FUNCTION INITIALIZE : BOOL
VAR_INPUT
END_VAR
VAR
	i : INT;
	GVL_IO: INT;
	SECTION2_DIG_INPUTS: INT;
	SECTION1_DIG_INPUTS: INT;
	JBOX_JBOX_GVL_LOGS: INT;
	NUM_TESTS_LOGGED: INT;
END_VAR


JBOX_GVL_LOGS.NUM_TESTS_LOGGED := 0;


JBOX_GVL_IO.SECTION1_DIG_INPUTS[0] := ADR(JBOX_GVL_IO.J7_24V_Up);
JBOX_GVL_IO.SECTION1_DIG_INPUTS[1] := ADR(JBOX_GVL_IO.J7_24V_Us);
JBOX_GVL_IO.SECTION1_DIG_INPUTS[2] := ADR(JBOX_GVL_IO.J8_24V_Up);
JBOX_GVL_IO.SECTION1_DIG_INPUTS[3] := ADR(JBOX_GVL_IO.J8_24V_Us);
JBOX_GVL_IO.SECTION1_DIG_INPUTS[4] := ADR(JBOX_GVL_IO.J1_24V_Up);
JBOX_GVL_IO.SECTION1_DIG_INPUTS[5] := ADR(JBOX_GVL_IO.J1_24V_Us);
JBOX_GVL_IO.SECTION1_DIG_INPUTS[6] := ADR(JBOX_GVL_IO.J2_24V_Up);
JBOX_GVL_IO.SECTION1_DIG_INPUTS[7] := ADR(JBOX_GVL_IO.J2_24V_Us);
JBOX_GVL_IO.SECTION1_DIG_INPUTS[8] := ADR(JBOX_GVL_IO.J3_24V_Up);
JBOX_GVL_IO.SECTION1_DIG_INPUTS[9] := ADR(JBOX_GVL_IO.J3_24V_Us);
JBOX_GVL_IO.SECTION1_DIG_INPUTS[10] := ADR(JBOX_GVL_IO.J4_24V_Up);
JBOX_GVL_IO.SECTION1_DIG_INPUTS[11] := ADR(JBOX_GVL_IO.J4_24V_Us);
JBOX_GVL_IO.SECTION1_DIG_INPUTS[12] := ADR(JBOX_GVL_IO.J5_24V_Up);
JBOX_GVL_IO.SECTION1_DIG_INPUTS[13] := ADR(JBOX_GVL_IO.J5_24V_Us);
JBOX_GVL_IO.SECTION1_DIG_INPUTS[14] := ADR(JBOX_GVL_IO.J6_24V_Up);
JBOX_GVL_IO.SECTION1_DIG_INPUTS[15] := ADR(JBOX_GVL_IO.J6_24V_Us);
JBOX_GVL_IO.SECTION1_DIG_INPUTS[16] := ADR(JBOX_GVL_IO.SF1_MF_CONTINUITY);
JBOX_GVL_IO.SECTION1_DIG_INPUTS[17] := ADR(JBOX_GVL_IO.SF2_MF_CONTINUITY);
JBOX_GVL_IO.SECTION1_DIG_INPUTS[18] := ADR(JBOX_GVL_IO.SF4_Pull_Station);
JBOX_GVL_IO.SECTION1_DIG_INPUTS[19] := ADR(JBOX_GVL_IO.SF6_MGT_CONTINUITY);
JBOX_GVL_IO.SECTION1_DIG_INPUTS[20] := ADR(JBOX_GVL_IO.SF8_MGT_CONTINUITY);
JBOX_GVL_IO.SECTION1_DIG_INPUTS[21] := ADR(JBOX_GVL_IO.JB_Door_Switch);
JBOX_GVL_IO.SECTION1_DIG_INPUTS[22] := ADR(JBOX_GVL_IO.JB_DCDCS_OK);
JBOX_GVL_IO.SECTION1_DIG_INPUTS[23] := ADR(JBOX_GVL_IO.JB_PSU1_OK);


JBOX_GVL_IO.SECTION2_DIG_INPUTS[0] := ADR(JBOX_GVL_IO.SF4_Pull_Station);
JBOX_GVL_IO.SECTION2_DIG_INPUTS[1] := ADR(JBOX_GVL_IO.JB_Door_Switch);
JBOX_GVL_IO.SECTION2_DIG_INPUTS[2] := ADR(JBOX_GVL_IO.JB_PSU2_OK);
JBOX_GVL_IO.SECTION2_DIG_INPUTS[3] := ADR(JBOX_GVL_IO.J7_24V_Up);
JBOX_GVL_IO.SECTION2_DIG_INPUTS[4] := ADR(JBOX_GVL_IO.J7_24V_Us);
JBOX_GVL_IO.SECTION2_DIG_INPUTS[5] := ADR(JBOX_GVL_IO.J8_24V_Up);
JBOX_GVL_IO.SECTION2_DIG_INPUTS[6] := ADR(JBOX_GVL_IO.J8_24V_Us);
JBOX_GVL_IO.SECTION2_DIG_INPUTS[7] := ADR(JBOX_GVL_IO.J1_24V_Up);
JBOX_GVL_IO.SECTION2_DIG_INPUTS[8] := ADR(JBOX_GVL_IO.J1_24V_Us);
JBOX_GVL_IO.SECTION2_DIG_INPUTS[9] := ADR(JBOX_GVL_IO.J2_24V_Up);
JBOX_GVL_IO.SECTION2_DIG_INPUTS[10] := ADR(JBOX_GVL_IO.J2_24V_Us);
JBOX_GVL_IO.SECTION2_DIG_INPUTS[11] := ADR(JBOX_GVL_IO.J3_24V_Up);
JBOX_GVL_IO.SECTION2_DIG_INPUTS[12] := ADR(JBOX_GVL_IO.J3_24V_Us);
JBOX_GVL_IO.SECTION2_DIG_INPUTS[13] := ADR(JBOX_GVL_IO.J4_24V_Up);
JBOX_GVL_IO.SECTION2_DIG_INPUTS[14] := ADR(JBOX_GVL_IO.J4_24V_Us);
JBOX_GVL_IO.SECTION2_DIG_INPUTS[15] := ADR(JBOX_GVL_IO.J5_24V_Up);
JBOX_GVL_IO.SECTION2_DIG_INPUTS[16] := ADR(JBOX_GVL_IO.J5_24V_Us);
JBOX_GVL_IO.SECTION2_DIG_INPUTS[17] := ADR(JBOX_GVL_IO.J6_24V_Up);
JBOX_GVL_IO.SECTION2_DIG_INPUTS[18] := ADR(JBOX_GVL_IO.J6_24V_Us);


INITIALIZE := TRUE;

END_FUNCTION

(* stored: Version 1.1.0.1, ProductVersion 3.1.4024.10
   POU INITIALIZE: Id {9eee4c6a-b7fe-4839-94e4-ff9f40c4ce0f}, SpecialFunc None *)
